// TIA Portal V16 export
// export: Created 2024-09-05T17:39:13.7826897Z, ExportSetting WithDefaults, DisplayName Totally Integrated Automation Portal, DisplayVersion V16 Update 6, DisplayName TIA Portal Version Control Interface, DisplayVersion V16 Update 2, DisplayName TIA Portal Openness, DisplayVersion V16 Update 6, DisplayName STEP 7 Professional, DisplayVersion V16 Update 6, DisplayName STEP 7 Safety, DisplayVersion V16, DisplayName WinCC Advanced, DisplayVersion V16 Update 6
DATA_BLOCK "Reader Parameters"   // DB300
{ S7_Optimized_Access := 'TRUE' }
VERSION : 0.1
// stored: AutoNumber false, DBAccessibleFromOPCUA true, IsOnlyStoredInLoadMemory false, IsRetainMemResEnabled false, IsWriteProtectedInAS false, MemoryReserve 100
   VAR
      Reader : Array[1.."MaxReader"] of "UDT_CognexReaders";
   END_VAR
BEGIN
   Reader[1].HW.In.AcquisitionStatus := 424;
   Reader[1].HW.In.ResultsStatus := 422;
   Reader[1].HW.In.SoftEventControl := 388;
   Reader[1].HW.In.ResultData := 386;
   Reader[1].HW.Out.AcquisitionControl := 434;
   Reader[1].HW.Out.ResultsControl := 423;
   Reader[1].HW.Out.SoftEventControl := 388;
   Reader[1].HW.Out.UserData := 387;
END_DATA_BLOCK
